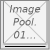
VISUALIZATION F_MainMenu_01  // 50x50
VAR_IN_OUT
	stMenuButton	: ST_HMIEButton_HMI;
END_VAR
    Image (3,0 44x44), image: ImagePool.01_Parameters
        OnMouseDown: execute { stMenuButton.bPushed := TRUE; }
    Line (5,46) (45,46), invisible if: not stMenuButton.bVisible or not stMenuButton.bActive, input disabled if: not stMenuButton.bEnable
END_VISUALIZATION

(* stored: Version 1.1.0.1
   Visu F_MainMenu_01: Id {93ac1001-74a3-01ec-0033-5a34129960ba} *)
